FUNCTION_BLOCK RequestQueueManager (* Ground-truth reference: elevator request arbitration (ported from the UAO curriculum's Elevator_DumbButtons exercise) *)
  (* Standard: 61499-2; Description: Educational reference, ported for the Meisterschulen am Ostbahnhof IEC 61499 training repository. Original design (c) nxtControl GmbH, from the UniversalAutomation.org 'IEC 61499: primer course' curriculum exercise Elevator_DumbButtons_EAE_Final.sln, IEC61499/RequestQueueManager.fbt - included here under the same educational-use terms as the rest of that curriculum. This port: Copyright (c) 2026 Meisterschulen am Ostbahnhof, EPL-2.0, https://www.eclipse.org/legal/epl-2.0/ *)
  (* Version 0.0, 2021-09-24, ferch, nxtControl GmbH, Original EAE/nxtControl design (Template), source: Elevator_DumbButtons_EAE_Final.sln *)
  (* Version 1.0, 2026-09-03, Franz Höpfinger, Meisterschulen am Ostbahnhof, Ported from EAE/nxtControl format (LibraryElement.dtd) to 4diac's FBType XSD: dropped EAE-only bookkeeping attributes (GUID, Configuration.FB.IDCounter, FBType.Basic.Algorithm.Order), added Type= on every Event (originally untyped) - interface, ECC, and all seven algorithms otherwise unchanged from the original. Found while searching the curriculum for ground truth on the Chain-of-Actions pattern (see ChainOfActionsPattern.md, 'Ground-truth reference' section) - a real, working example combining REQ/CNF service-style events with chain-style sequencing. NOTE: this FB's own REQ is unrelated to TrueUntil.fbt's still-open REQ-vs-TRIGGER question in the same folder - different block, does not resolve that ambiguity, just a topically similar precedent *)
  (* Version 1.1, 2026-09-03, Franz Höpfinger, Meisterschulen am Ostbahnhof, PR #160 review feedback: INIT/INITO must be Type=EInit (were Type=Event) - fixed, With-Var lists unchanged *)
  (* Version 1.2, 2026-09-03, Franz Höpfinger, Meisterschulen am Ostbahnhof, PR #160 review feedback (coderabbitai): the INIT algorithm declared Floor_Req_*/Cabin_Req_* as With-Vars but never read them, so a request already active at deployment was ignored until a later REQ - fixed by latching requests[]/pending_reqs from the INIT snapshot, same as READ_REQS does. A genuine behavior fix, not a faithfulness-preserving port choice like the other two VersionInfo entries above *)
  PACKAGE Meins::DesingPatterns::ChainOfActionsPattern;
  (* Documentation:
  Ground-truth reference, not a Vyatkin Module 6 slide pattern. Ported as-is (same interface, same ECC, same seven algorithms) from the UniversalAutomation.org "IEC 61499: primer course" curriculum exercise Elevator_DumbButtons_EAE_Final.sln (IEC61499/RequestQueueManager.fbt, original format: EAE/nxtControl LibraryElement.dtd), found while searching that curriculum's Downloads export for material relevant to this repo's Chain of Actions pattern implementation.
   Real elevator-request arbitrator: a classic SCAN-disk-style sweep (DETERMINE) picks the next pending floor in the current sweep direction, sends MOVE_ELEVATOR, waits for DONE_MOVE, opens the door (DOOR_IN, with a first CNF acknowledging arrival), waits for DONE_DOOR, then closes it and clears the request (a second CNF confirming completion) before returning to WAITING. Combines this repo's two adjacent ideas in one real, working block: Chain-of-Actions-style sequencing (a handful of small states forming one linear worklist loop) and REQ/CNF service-style events (matching the vocabulary also seen in the Handshake pattern and the slide-47 message-exchange example) - worth comparing against TrueUntil.fbt in this same folder - though this block's own REQ is unrelated to TrueUntil.fbt's still-open REQ-vs-TRIGGER question, it does not resolve that ambiguity.
   Kept faithful to the original on purpose, including its quirks: no QI/QO initialization qualifier (this repo's usual Init/Initialized/DeInit convention does not apply here - `INIT` is just a regular event that happens to carry the initial request snapshot), and CNF firing twice per serviced request with different payload each time (arrival vs. completion) rather than using two distinct event names.
  *)
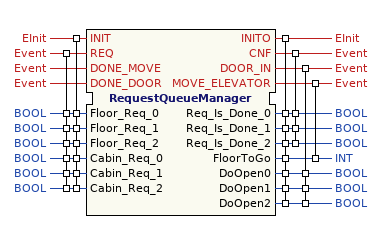
  EVENT_INPUT
    INIT : EInit WITH Floor_Req_0, Floor_Req_1, Floor_Req_2, Cabin_Req_0, Cabin_Req_1, Cabin_Req_2; (* Initialization Request - carries the initial request snapshot, not the repo's usual QI qualifier *)
    REQ WITH Floor_Req_0, Floor_Req_1, Floor_Req_2, Cabin_Req_0, Cabin_Req_1, Cabin_Req_2; (* Normal Execution Request: a floor or cabin button was pressed *)
    DONE_MOVE; (* The elevator actuator confirms it reached FloorToGo *)
    DONE_DOOR; (* The door actuator confirms the open/close cycle is done *)
  END_EVENT
  EVENT_OUTPUT
    INITO : EInit WITH Req_Is_Done_0, Req_Is_Done_1, Req_Is_Done_2, FloorToGo, DoOpen0, DoOpen1, DoOpen2; (* Initialization Confirm *)
    CNF WITH Req_Is_Done_0, Req_Is_Done_1, Req_Is_Done_2; (* Execution Confirmation - fired twice per serviced request: once on arrival (door opens), once on completion (door closes) *)
    DOOR_IN WITH DoOpen0, DoOpen1, DoOpen2; (* Command the door actuator to open *)
    MOVE_ELEVATOR WITH FloorToGo; (* Command the elevator actuator to move to FloorToGo *)
  END_EVENT
  VAR_INPUT
    Floor_Req_0 : BOOL;
    Floor_Req_1 : BOOL;
    Floor_Req_2 : BOOL;
    Cabin_Req_0 : BOOL;
    Cabin_Req_1 : BOOL;
    Cabin_Req_2 : BOOL;
  END_VAR
  VAR_OUTPUT
    Req_Is_Done_0 : BOOL;
    Req_Is_Done_1 : BOOL;
    Req_Is_Done_2 : BOOL;
    FloorToGo : INT;
    DoOpen0 : BOOL;
    DoOpen1 : BOOL;
    DoOpen2 : BOOL;
  END_VAR
  VAR
    up_direction : BOOL; (* SCAN-style sweep direction: TRUE = scanning floors upward *)
    index : INT; (* Floor currently being scanned/serviced *)
    do_request : BOOL; (* DETERMINE loop exit flag: a pending request was found at index *)
    pending_reqs : BOOL; (* TRUE while any floor/cabin request is still outstanding *)
    requests : ARRAY [0..2] OF BOOL := [3(FALSE)]; (* Per-floor outstanding-request flags (floor OR cabin button) *)
  END_VAR
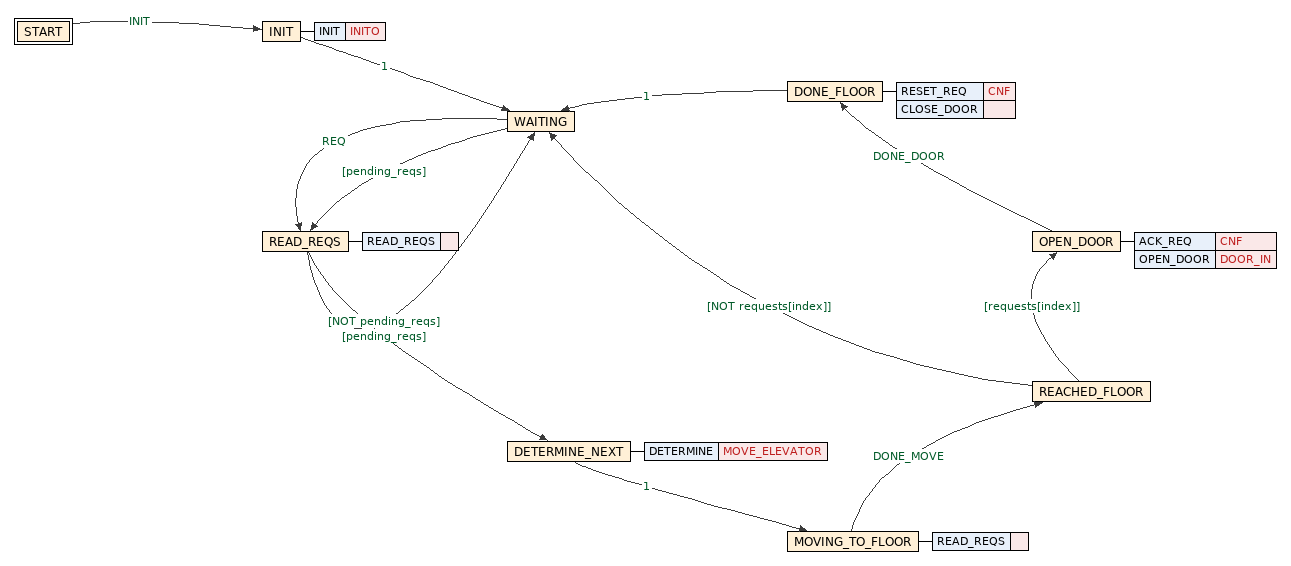
  EC_STATES
    START; (* Initial State *)
    INIT : INIT -> INITO; (* Initialization *)
    WAITING; (* Idle, no move in progress *)
    READ_REQS : READ_REQS; (* Latch Floor_Req_*/Cabin_Req_* into the requests array *)
    DETERMINE_NEXT : DETERMINE -> MOVE_ELEVATOR; (* SCAN-style sweep to the next pending floor *)
    MOVING_TO_FLOOR : READ_REQS; (* Waiting for the elevator actuator *)
    REACHED_FLOOR; (* Arrived at index: decide whether to open the door *)
    OPEN_DOOR : ACK_REQ -> CNF, OPEN_DOOR -> DOOR_IN; (* Ack the request, command the door open *)
    DONE_FLOOR : RESET_REQ -> CNF, CLOSE_DOOR; (* Door confirmed open/closed: clear the request, close the door *)
  END_STATES
  EC_TRANSITIONS
    START TO INIT := INIT;
    INIT TO WAITING := 1;
    WAITING TO READ_REQS := REQ;
    READ_REQS TO WAITING := [NOT pending_reqs];
    READ_REQS TO DETERMINE_NEXT := [pending_reqs];
    DETERMINE_NEXT TO MOVING_TO_FLOOR := 1;
    MOVING_TO_FLOOR TO REACHED_FLOOR := DONE_MOVE;
    REACHED_FLOOR TO OPEN_DOOR := [requests[index]];
    REACHED_FLOOR TO WAITING := [NOT requests[index]];
    OPEN_DOOR TO DONE_FLOOR := DONE_DOOR;
    DONE_FLOOR TO WAITING := 1;
    WAITING TO READ_REQS := [pending_reqs];
  END_TRANSITIONS
  ALGORITHM INIT IN ST: (* Reset all outputs and internal state, latching any request already present at deployment *)
Req_Is_Done_0 := FALSE;
Req_Is_Done_1 := FALSE;
Req_Is_Done_2 := FALSE;
// Initialize the elevator at 0 floor on startup
FloorToGo := 0;
DoOpen0 := FALSE;
DoOpen1 := FALSE;
DoOpen2 := FALSE;
// Internal variables
up_direction := TRUE;
index := -1;
do_request := FALSE;
// Latch the request snapshot carried by INIT itself (fixes: an initial
// request was previously ignored until a later REQ event)
requests[0] := Floor_Req_0 OR Cabin_Req_0;
requests[1] := Floor_Req_1 OR Cabin_Req_1;
requests[2] := Floor_Req_2 OR Cabin_Req_2;
pending_reqs := requests[0] OR requests[1] OR requests[2];
  END_ALGORITHM
  ALGORITHM READ_REQS IN ST: (* Latch the button inputs into the requests array *)
requests[0] := Floor_Req_0 OR Cabin_Req_0;
requests[1] := Floor_Req_1 OR Cabin_Req_1;
requests[2] := Floor_Req_2 OR Cabin_Req_2;
pending_reqs := requests[0] OR requests[1] OR requests[2];
  END_ALGORITHM
  ALGORITHM DETERMINE IN ST: (* SCAN elevator algorithm: sweep up then down, stop at the next pending floor *)
do_request := FALSE;
WHILE NOT do_request DO
	// Change index direction
	IF index = 2 THEN
		up_direction := FALSE;
	ELSIF index = 0 THEN
		up_direction := TRUE;
	END_IF;
	// Increment/Decrement index consequently to direction
	IF up_direction THEN
		index := index + 1;
	ELSE
		index := index - 1;
	END_IF;
	// Check whether there is a pending request in this index
	IF requests[index] THEN
		do_request := TRUE;
		// Output the floor_to_go to the ElevatorMoveControl
		FloorToGo := index;
	END_IF;
END_WHILE;
  END_ALGORITHM
  ALGORITHM OPEN_DOOR IN ST: (* Command the door at the current index open *)
IF index = 0 THEN
	DoOpen0 := TRUE;
ELSIF index = 1 THEN
	DoOpen1 := TRUE;
ELSE
	DoOpen2 := TRUE;
END_IF;
  END_ALGORITHM
  ALGORITHM RESET_REQ IN ST: (* Clear the serviced request and recompute pending_reqs *)
// Reset all output variables (only one was TRUE, but for simplicity all are cleared)
Req_Is_Done_0 := FALSE;
Req_Is_Done_1 := FALSE;
Req_Is_Done_2 := FALSE;
// Clear the attended request on the request array
requests[index] := FALSE;
// Update pending_requests variable
pending_reqs := requests[0] OR requests[1] OR requests[2];
  END_ALGORITHM
  ALGORITHM CLOSE_DOOR IN ST: (* Command all doors closed *)
// For simplicity, all of them are reset to FALSE
DoOpen0 := FALSE;
DoOpen1 := FALSE;
DoOpen2 := FALSE;
  END_ALGORITHM
  ALGORITHM ACK_REQ IN ST: (* Mark the request at the current index as being handled *)
IF index = 0 THEN
	Req_Is_Done_0 := TRUE;
ELSIF index = 1 THEN
	Req_Is_Done_1 := TRUE;
ELSE
	Req_Is_Done_2 := TRUE;
END_IF;
  END_ALGORITHM
END_FUNCTION_BLOCK
